(* IEC 61131-3 sources: automatic-screwdriver-line/src/Plant_Simulation, 2 files *)

(* ---- IO_Simulation.st ---- *)
// Generated from Automatic_ScrewDriver_Line.xml by tools/export_st.py - do not edit.
// The CODESYS project is the source of truth.

{attribute 'qualified_only'}
VAR_GLOBAL
	// Mover
	// Outputs: PLC to Machine
	MoverEnable : BOOL;
	MoverExecuteFor : BOOL;
	MoverExecuteBac : BOOL;
	MoverActPos : REAL;   // Inputs: Machine to PLC
	MoverReady : BOOL;
	// Z Axis
	// Outputs: PLC to Machine
	zValve : BOOL;
	zDown : BOOL;   // Inputs: Machine to PLC
	ScrewEngaged : BOOL;
	ScrewReleased : BOOL;
	// Spindle
	// Outputs: PLC to Machine
	SpindleEnable : BOOL;
	SpindleExecute : BOOL;
	SpindleExecuteTime : TIME;
	SpindleReady : BOOL;   // Inputs: Machine to PLC
	SpindleDone : BOOL;
	SimFail_ScrewEngaged : BOOL;   // Z axis rises but the bit never engages the screw
	SimFail_ScrewReleased : BOOL;   // bit stays stuck in the screw head
	SimFail_SpindleDone : BOOL;   // spindle never reports completion
	SimFail_MoverReady : BOOL;   // drive never confirms torque
	SimFail_MoverBlocked : BOOL;   // axis is commanded but does not move
END_VAR

(* ---- PRG_PlantSim.st ---- *)
// Generated from Automatic_ScrewDriver_Line.xml by tools/export_st.py - do not edit.
// The CODESYS project is the source of truth.

PROGRAM PRG_PlantSim
VAR
	_Increment : REAL := 1;
	_ZAxisMovingTimeUp : TON;
	_ZAxisMovingTimeDown : TON;
	_SpindleMovingTime : TON;
END_VAR

// Conveyor
IO_Simulation.MoverReady := IO_Simulation.MoverEnable
                                   AND NOT IO_Simulation.SimFail_MoverReady;
IF IO_Simulation.MoverExecuteFor AND IO_Simulation.MoverEnable
   AND NOT IO_Simulation.SimFail_MoverBlocked THEN
    IO_Simulation.MoverActPos := IO_Simulation.MoverActPos + _Increment;
ELSIF IO_Simulation.MoverExecuteBac AND IO_Simulation.MoverEnable
   AND NOT IO_Simulation.SimFail_MoverBlocked THEN
    IO_Simulation.MoverActPos := IO_Simulation.MoverActPos - _Increment;
END_IF

// Z Axis
_ZAxisMovingTimeUp(IN := IO_Simulation.zValve, PT := T#1S);
IO_Simulation.ScrewEngaged := _ZAxisMovingTimeUp.Q
                                     AND NOT IO_Simulation.SimFail_ScrewEngaged;
_ZAxisMovingTimeDown(IN := NOT IO_Simulation.zValve, PT := T#1S);
IO_Simulation.ScrewReleased := _ZAxisMovingTimeDown.Q
                                      AND NOT IO_Simulation.SimFail_ScrewReleased;
// zDown is not filtered: the cylinder physically retracts even if the bit stays engaged
IO_Simulation.zDown := _ZAxisMovingTimeDown.Q;

// Spindle
IO_Simulation.SpindleReady := IO_Simulation.SpindleEnable;
_SpindleMovingTime(IN := IO_Simulation.SpindleExecute
                         AND IO_Simulation.SpindleEnable,
                   PT := IO_Simulation.SpindleExecuteTime);
IO_Simulation.SpindleDone := _SpindleMovingTime.Q
                                    AND NOT IO_Simulation.SimFail_SpindleDone;

END_PROGRAM
